(* IEC 61131-3 sources: TIA2AX/tests/V18/test_projects/expected/HW_DiscoverGroups/PLC_6, 7 files *)

(* ---- HwIdentifiers.st ---- *)
TYPE
	HwIdentifiers : WORD
	(
		PLC_6_Rail_0 :=	WORD#256,
		PLC_6 :=	WORD#48,
		PLC_6_Card_reader_writer_1 :=	WORD#51,
		PLC_6_CPU_display_1 :=	WORD#54,
		PLC_6_OPC_UA_1 :=	WORD#117,
		PLC_6_PROFINET_interface_1 :=	WORD#64,
		PLC_6_PROFINET_interface_1_Port_1 :=	WORD#65,
		PLC_6_PROFINET_interface_1_Port_2 :=	WORD#66,
		NONE:= WORD#0
	);
END_TYPE

(* ---- HwInputs.st ---- *)
TYPE
	HwInputs : STRUCT
	END_STRUCT;
END_TYPE

(* ---- HwOutputs.st ---- *)
TYPE
	HwOutputs : STRUCT
	END_STRUCT;
END_TYPE

(* ---- PlcInputs.st ---- *)
TYPE
	PlcInputs : STRUCT
	END_STRUCT;
END_TYPE

(* ---- PlcOutputs.st ---- *)
TYPE
	PlcOutputs : STRUCT
	END_STRUCT;
END_TYPE

(* ---- CopyInputs.st ---- *)
FUNCTION CopyInputs
	VAR_EXTERNAL
		HwInputs : HwInputs;
		PlcInputs : PlcInputs;
	END_VAR
END_FUNCTION

(* ---- CopyOutputs.st ---- *)
FUNCTION CopyOutputs
	VAR_EXTERNAL
		HwOutputs : HwOutputs;
		PlcOutputs : PlcOutputs;
	END_VAR
END_FUNCTION
